{attribute addProperty BoxType "KL9900-0057"}
{attribute addProperty Id "Channel_1Channel_646A3FAD00"}
{attribute addProperty CRC "3969081270"}
{attribute addProperty SizeInBites "0"}
{attribute addProperty SizeInBytes "0"}
TYPE KL_EC935FB6 :
STRUCT
	{attribute addProperty Name "Channel_1"}
	Channel_1 : Channel_646A3FAD;
END_STRUCT
END_TYPE

(* stored: Version 1.2.0.0, ProductVersion 3.1.4024.9
   DUT KL_EC935FB6: Id {655debc6-b675-40fb-b055-f7fe10f09b80} *)
